# B&R Automation Studio project Binary-to-BCD
Automation Studio 4.9.2.46

## Configuration Config1

CPU X20CP1586, AutomationRuntime C4.90, Build 4.1.2, Vc V4.72.2

### Hardware
```
X20CP1586 : X20CP1586 v1.8.1.0
  Connector IF2:
    ActivateDevice = 1
  Simulation = 1
```

## Logical view

### Global.var
```iecst
VAR
	(* Binary - input *)
	B3 : BOOL;
	B2 : BOOL;
	B1 : BOOL;
	B0 : BOOL;

	(* BCD - output *)
	D4 : BOOL;
	D3 : BOOL;
	D2 : BOOL;
	D1 : BOOL;
	D0 : BOOL;

	(* Helper variables *)
	H09 : BOOL; (* input in 0-9 *)
	H1213 : BOOL; (* input in 12-13 *)
	H89 : BOOL; (* input in 8-9 *)
END_VAR
```

### Program Logical/Program

#### Cyclic.ld
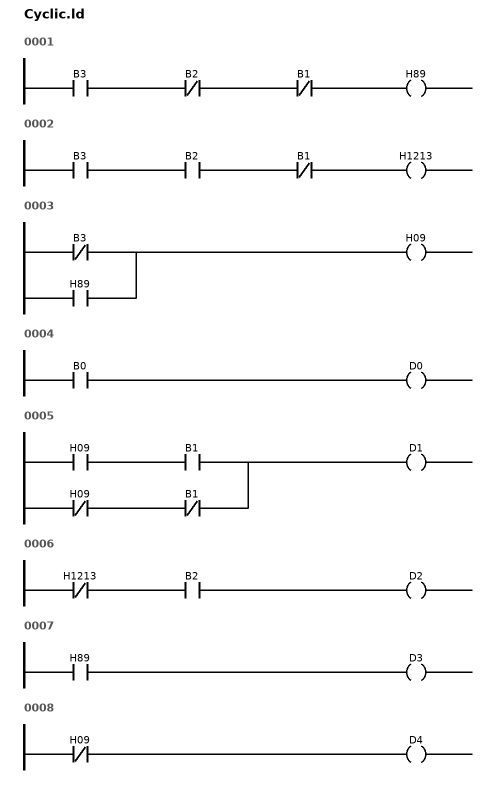
Ladder, written as Structured Text:
```iecst
PROGRAM _CYCLIC
(* Network 1 *)
H89 := B3 AND NOT B2 AND NOT B1;

(* Network 2 *)
H1213 := B3 AND B2 AND NOT B1;

(* Network 3 *)
H09 := NOT B3 OR H89;

(* Network 4 *)
D0 := B0;

(* Network 5 *)
D1 := (H09 AND B1) OR (NOT H09 AND NOT B1);

(* Network 6 *)
D2 := NOT H1213 AND B2;

(* Network 7 *)
D3 := H89;

(* Network 8 *)
D4 := NOT H09;
END_PROGRAM
```
